FUNCTION_BLOCK LREAL_Param
VAR_INPUT PERSISTENT
	val			: LREAL;
END_VAR

END_FUNCTION_BLOCK

(* stored: Version 1.1.0.1
   POU LREAL_Param: Id {d6017903-1f79-4c2a-8e02-b33751064f9a}, SpecialFunc None *)
